SUBAPPLICATION Uebung_212 (* Standard IEC 61131-3 FB_CTU_LINT (Vorwärtszähler, LINT) mit Terminal-Ausgabe *)
  (* Standard: 61131-3; Description: Copyright (c) 2026 Meisterschulen am Ostbahnhof This program and the accompanying materials are made available under the terms of the Eclipse Public License 2.0 which is available at https://www.eclipse.org/legal/epl-2.0/ SPDX-License-Identifier: EPL-2.0 *)
  (* Version 1.1, 2026-04-21, Franz Höpfinger, Meisterschulen am Ostbahnhof, Added terminal output for counter value *)
  (* Version 1.0, 2026-04-20, Franz Höpfinger, Meisterschulen am Ostbahnhof, initial API and implementation (IEC 61131-3 version) *)
  PACKAGE Uebungen;
  IMPORT Uebungen::const::UT::DefaultPool::OutputNumber_N1;
  IMPORT logiBUS::io::DI::logiBUS_DI::Input_I1;
  IMPORT logiBUS::io::DI::logiBUS_DI::Input_I2;
  IMPORT logiBUS::io::DQ::logiBUS_DO::Output_Q1;
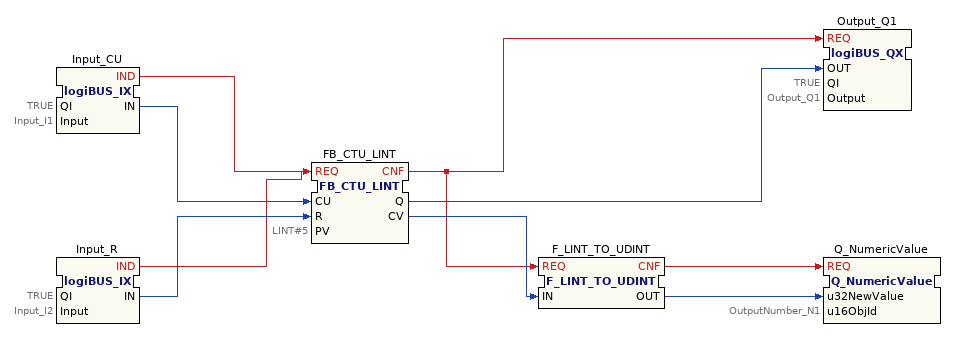
  FBS
    FB_CTU_LINT : iec61131::counters::FB_CTU_LINT(PV := LINT#5);
    Input_CU : logiBUS::io::DI::logiBUS_IX(QI := TRUE, Input := Input_I1);
    Input_R : logiBUS::io::DI::logiBUS_IX(QI := TRUE, Input := Input_I2);
    Output_Q1 : logiBUS::io::DQ::logiBUS_QX(QI := TRUE, Output := Output_Q1);
    Q_NumericValue : isobus::UT::Q::Q_NumericValue(u16ObjId := OutputNumber_N1);
    F_LINT_TO_UDINT : iec61131::conversion::F_LINT_TO_UDINT;
  END_FBS
  EVENT_CONNECTIONS
    Input_CU.IND TO FB_CTU_LINT.REQ;
    Input_R.IND TO FB_CTU_LINT.REQ;
    FB_CTU_LINT.CNF TO Output_Q1.REQ;
    FB_CTU_LINT.CNF TO F_LINT_TO_UDINT.REQ;
    F_LINT_TO_UDINT.CNF TO Q_NumericValue.REQ;
  END_CONNECTIONS
  DATA_CONNECTIONS
    Input_CU.IN TO FB_CTU_LINT.CU;
    Input_R.IN TO FB_CTU_LINT.R;
    FB_CTU_LINT.Q TO Output_Q1.OUT;
    FB_CTU_LINT.CV TO F_LINT_TO_UDINT.IN;
    F_LINT_TO_UDINT.OUT TO Q_NumericValue.u32NewValue;
  END_CONNECTIONS
END_SUBAPPLICATION
